Fanuc TP program (LS listing): w1_chuck_opn.ls

/PROG  W1_CHUCK_OPN
/ATTR
OWNER		= MNEDITOR;
COMMENT		= "";
PROG_SIZE	= 398;
CREATE		= DATE 19-03-20  TIME 13:53:46;
MODIFIED	= DATE 19-03-20  TIME 13:55:22;
FILE_NAME	= W1_CHUCK;
VERSION		= 0;
LINE_COUNT	= 15;
MEMORY_SIZE	= 874;
PROTECT		= READ_WRITE;
TCD:  STACK_SIZE	= 0,
      TASK_PRIORITY	= 50,
      TIME_SLICE	= 0,
      BUSY_LAMP_OFF	= 0,
      ABORT_REQUEST	= 0,
      PAUSE_REQUEST	= 0;
DEFAULT_GROUP	= 1,*,*,*,*;
CONTROL_CODE	= 00000000 00000000;
/APPL
/MN
   1:  DO[43:W1_Chuck_Close]=OFF ;
   2:  DO[42:W1_Chuck_Open]=ON ;
   3:  WAIT   1.00(sec) ;
   4:   ;
   5:  $WAITTMOUT=200 ;
   6:  WAIT (DI[49:W1_Chuck_Opened]) TIMEOUT,LBL[1] ;
   7:   ;
   8:   ;
   9:  END ;
  10:  LBL[1] ;
  11:  MESSAGE[...] ;
  12:  MESSAGE[AMERIKANER] ;
  13:  MESSAGE[NIJE OTVORIO] ;
  14:  WAIT (DI[49:W1_Chuck_Opened])    ;
  15:  END ;
/POS
/END
